{attribute 'GeneratedUsingTerminal: EL3024-0000-0019'}
{attribute addProperty BoxType "EL3024-0000-0019"}
{attribute addProperty Id "AdsAddrAT %I*.TcoAmsAddr0StateAT %I*UINT2"}
{attribute addProperty CRC "2493615966"}
{attribute addProperty Size "2"}
TYPE InfoData_94A18F5E :
STRUCT
	{attribute addProperty Name "AdsAddr"}
	AdsAddr AT %I* : .TcoAmsAddr;
	{attribute addProperty Name "State"}
	State AT %I* : UINT;
END_STRUCT
END_TYPE
